FUNCTION_BLOCK eye
VAR_OUTPUT
    I: ARRAY [0..8] OF LREAL;
END_VAR
VAR_TEMP
    b_i: DINT;
END_VAR

FOR b_i := 0 TO 8 DO 
    I[b_i] := 0.0;
END_FOR;
I[0] := 1.0;
I[4] := 1.0;
I[8] := 1.0;

END_FUNCTION_BLOCK

(* stored: Version 1.1.0.1, ProductVersion 3.1.4024.12
   POU eye: Id {ed62f816-13c3-4ac9-9b30-2738105912f0}, SpecialFunc None *)
